TEXTLIST PDU_Breaker_Status
  0 = 'Open'
  1 = 'Closed'
   = ''
END_TEXTLIST

(* stored: Version 1.1.0.1, ProductVersion 3.1.4024.12
   TextList PDU_Breaker_Status: Id {91ec6886-174b-42e9-b284-9d5982b58ef7} *)
